FUNCTION_BLOCK DigitalInputNC
VAR_INPUT
	input				: BOOL;
END_VAR
VAR_OUTPUT
	isActive			: BOOL;
	isNotActive			: BOOL;
	inputHasRisingEdge	: BOOL;
	inputHasFallingEdge	: BOOL;
END_VAR
VAR
	edgeR				: r_trig;
	edgeF				: f_trig;
END_VAR

isActive				:= NOT input;
isNotActive				:= input;

edgeR(CLK:=isActive, Q=>inputHasRisingEdge);
edgeF(CLK:=NOT isActive, Q=>inputHasFallingEdge);

END_FUNCTION_BLOCK

(* stored: Version 1.1.0.1
   POU DigitalInputNC: Id {9c561f21-f254-46a2-bf63-c42558e21c02}, SpecialFunc None *)
